(* IEC 61131-3 sources: WarwickBoringPLC/MaterialExtraction, 2 files *)

(* ---- meFeederPumpControl.st ---- *)
FUNCTION_BLOCK meFeederPumpControl
VAR_INPUT
END_VAR
VAR_OUTPUT
END_VAR
VAR
	feederPumpClock : CLK; // Feeder pump clock
	onPeriod : TIME;
	offPeriod : TIME;
END_VAR

onPeriod = REAL_TO_TIME(TIME_TO_REAL(meGVL.meFeederPumpPeriod) * meFeederPumpDuty); //get on period
offPeriod = REAL_TO_TIME(TIME_TO_REAL(meGVL.meFeederPumpPeriod) - onPeriod); //get off period

feederPumpClock(EN:= meGVL.meFeederPumpEnabled AND meGVL.meFeederPumpUserEnabled, ON_PERIOD:= onPeriod, OFF_PERIOD:= offPeriod, Q=> meGVL.meFeederPumpAutoPower); //TODO - change on/off period to correct values

// If feeder pump is not enabled, the power off
IF NOT meGVL.meFeederPumpEnabled OR NOT meGVL.meFeederPumpUserEnabled THEN
	// Disable
	meGVL.mePowerFeederPump := FALSE;
ELSE
	// If auto mode
	IF meGVL.meFeederPumpAutoControlEnabled THEN
		meGVL.mePowerFeederPump := meGVL.meFeederPumpAutoPower;
	// Else in manual mode
	ELSE
		meGVL.mePowerFeederPump := meGVL.meFeederPumpManualPower;
	END_IF
END_IF

// Assign feeder pump contactor
mGVL.feederPumpContactor := meGVL.mePowerFeederPump;

(* ---- MaterialExtraction.st ---- *)
PROGRAM MaterialExtraction
VAR
	consumptionMeterLogic : meConsumption;
	feederPumpControlLogic : meFeederPumpControl;
END_VAR

// **********************************************************************
// ** VERSION 1.0.0 - Aaron 29/01/23**
// Carries out Material Extraction logic
//
// Changelog:
// - Added ME flowmeter
// **********************************************************************

consumptionMeterLogic();
feederPumpControlLogic();

// #############################
// ### 1P Machine Power C12  ###
// #############################
// control for ME 1 Phase - polymer pump, polymer mixerhttps://www.sparkfun.com/datasheets/Sensors/Biometric/MQ-4.pdf
CASE systemGVL.systemState OF
	SYSTEM_STATE.STARTING, SYSTEM_STATE.RUNNING, UNSUSPENDING:
		meGVL.me1PMachineEnabled := TRUE; //polymer pump & mixer start
	ELSE
		meGVL.me1PMachineEnabled := FALSE; //polymer pump & mixer stop
END_CASE

// ####################
// ### Feeder Pump  ###
// ####################
// control for contactor of feeder pump
CASE systemGVL.systemState OF
	SYSTEM_STATE.STARTING, SYSTEM_STATE.RUNNING, SYSTEM_STATE.UNSUSPENDING:
		meGVL.meFeederPumpEnabled := TRUE; //feeder pump enabled
	ELSE
		meGVL.meFeederPumpEnabled := FALSE; //feeder pump disabled
END_CASE

// ##############################
// ### Suction Pump VFD Power ###
// ##############################
// control for contactor of suction pump VFD
CASE systemGVL.systemState OF
	SYSTEM_STATE.STARTING, SYSTEM_STATE.RUNNING, SYSTEM_STATE.SUSPENDING,
	SYSTEM_STATE.SUSPENDED, SYSTEM_STATE.UNSUSPENDING:
		meGVL.meSuctionPumpContactorEnabled := TRUE; //suction pump contactor enabled
	ELSE
		meGVL.meSuctionPumpContactorEnabled := FALSE; //suction pump contactor disabled
END_CASE

// ####################
// ### VFD Control  ###
// ####################
// control for run/stop of suction
// actively digging - running, unsuspending, starting
CASE systemGVL.systemState OF
	SYSTEM_STATE.STARTING, SYSTEM_STATE.RUNNING, UNSUSPENDING:
		meGVL.meSuctionPumpVFDEnabled := TRUE; //VFD start
	ELSE
		meGVL.meSuctionPumpVFDEnabled := FALSE; //VFD stop
END_CASE
